PROGRAM LogicAndCounters

END_PROGRAM

(* stored: Version 1.1.0.1
   POU LogicAndCounters: Id {b3940d90-3391-4326-991f-f728b27834e0}, SpecialFunc None *)
